// TIA Portal V17 export
// export: Created 2022-07-20T06:59:51.7556163Z, ExportSetting WithDefaults, DisplayName Totally Integrated Automation Portal, DisplayVersion V17, DisplayName TIA Portal Openness, DisplayVersion V17, DisplayName TIA Portal Version Control Interface, DisplayVersion V17, DisplayName SINAMICS Startdrive Advanced, DisplayVersion V17, DisplayName SINAMICS Startdrive G130, G150, S120, S150, SINAMICS MV, S210, DisplayVersion V17, DisplayName SINAMICS Startdrive G110M, G120, G120C, G120D, G120P, G115D, DisplayVersion V17, DisplayName STEP 7 Professional, DisplayVersion V17, DisplayName STEP 7 Safety, DisplayVersion V17, DisplayName WinCC Advanced, DisplayVersion V17
FUNCTION_BLOCK "FB10067_IperPrintingInkCircuitGen2"   // FB10067, LAD
{ S7_Optimized_Access := 'TRUE' }
VERSION : 0.1
// stored: AutoNumber false, IsIECCheckEnabled false, IsRetainMemResEnabled false, MemoryReserve 100, SetENOAutomatically false, UDAEnableTagReadback false
   VAR_INPUT
      Acknowledge : Bool;
      DegassingSystem_RisingInkSensor : Bool;
      Sensor1_Value { ExternalAccessible := 'False'; ExternalVisible := 'False'; ExternalWritable := 'False'} : Int;
      Sensor1_HighErrorThreshold { ExternalAccessible := 'False'; ExternalVisible := 'False'; ExternalWritable := 'False'} : Real;
      Sensor1_HighWarningThreshold { ExternalAccessible := 'False'; ExternalVisible := 'False'; ExternalWritable := 'False'} : Real;
      Sensor1_LowWarningThreshold { ExternalAccessible := 'False'; ExternalVisible := 'False'; ExternalWritable := 'False'} : Real;
      Sensor1_LowErrorThreshold { ExternalAccessible := 'False'; ExternalVisible := 'False'; ExternalWritable := 'False'} : Real;
      Sensor2_Value { ExternalAccessible := 'False'; ExternalVisible := 'False'; ExternalWritable := 'False'} : Int;
      Sensor2_HighErrorThreshold { ExternalAccessible := 'False'; ExternalVisible := 'False'; ExternalWritable := 'False'} : Real;
      Sensor2_HighWarningThreshold { ExternalAccessible := 'False'; ExternalVisible := 'False'; ExternalWritable := 'False'} : Real;
      Sensor2_LowWarningThreshold { ExternalAccessible := 'False'; ExternalVisible := 'False'; ExternalWritable := 'False'} : Real;
      Sensor2_LowErrorThreshold { ExternalAccessible := 'False'; ExternalVisible := 'False'; ExternalWritable := 'False'} : Real;
      BarrelWS_RawValue { ExternalAccessible := 'False'; ExternalVisible := 'False'; ExternalWritable := 'False'} : Int;
      BarrelWS_CalibrationValue_1 { ExternalAccessible := 'False'; ExternalVisible := 'False'; ExternalWritable := 'False'} : Real;
      BarrelWS_CalibrationValue_2 { ExternalAccessible := 'False'; ExternalVisible := 'False'; ExternalWritable := 'False'} : Real;
      BarrelWS_LowWarningThreshold { ExternalAccessible := 'False'; ExternalVisible := 'False'; ExternalWritable := 'False'} : Real;
      BarrelWS_HighWarningThreshold { ExternalAccessible := 'False'; ExternalVisible := 'False'; ExternalWritable := 'False'} : Real;
      BarrelWS_LowErrorThreshold { ExternalAccessible := 'False'; ExternalVisible := 'False'; ExternalWritable := 'False'} : Real;
      BarrelWS_HighErrorThreshold { ExternalAccessible := 'False'; ExternalVisible := 'False'; ExternalWritable := 'False'} : Real;
      Tank1_ReachLevel { ExternalAccessible := 'False'; ExternalVisible := 'False'; ExternalWritable := 'False'} : Real;
      Tank1_RegulationLevel { ExternalAccessible := 'False'; ExternalVisible := 'False'; ExternalWritable := 'False'} : Real;
      Tank2_ReachLevel { ExternalAccessible := 'False'; ExternalVisible := 'False'; ExternalWritable := 'False'} : Real;
      Tank2_RegulationLevel { ExternalAccessible := 'False'; ExternalVisible := 'False'; ExternalWritable := 'False'} : Real;
      SystemPressurized { ExternalAccessible := 'False'; ExternalVisible := 'False'; ExternalWritable := 'False'} : Bool;
      SystemDepressurized { ExternalAccessible := 'False'; ExternalVisible := 'False'; ExternalWritable := 'False'} : Bool;
   END_VAR
   VAR_OUTPUT
      DegassingSystem_SolenoidValve : Bool;
      DegassingSystem_RisingInkError : Bool;
      ActivePump { ExternalAccessible := 'False'; ExternalVisible := 'False'; ExternalWritable := 'False'} : Bool;
      PumpDirection { ExternalAccessible := 'False'; ExternalVisible := 'False'; ExternalWritable := 'False'} : Bool;
      ActiveGeneralSolenoid { ExternalAccessible := 'False'; ExternalVisible := 'False'; ExternalWritable := 'False'} : Bool;
      ActiveFillingSolenoid_1 { ExternalAccessible := 'False'; ExternalVisible := 'False'; ExternalWritable := 'False'} : Bool;
      ActiveFillingSolenoid_2 { ExternalAccessible := 'False'; ExternalVisible := 'False'; ExternalWritable := 'False'} : Bool;
      BarrelWS_CalibrationStatus_1 { ExternalAccessible := 'False'; ExternalVisible := 'False'; ExternalWritable := 'False'} : Bool;
      BarrelWS_CalibrationStatus_2 { ExternalAccessible := 'False'; ExternalVisible := 'False'; ExternalWritable := 'False'} : Bool;
      BarrelWS_LowWarningThresholdReached { ExternalAccessible := 'False'; ExternalVisible := 'False'; ExternalWritable := 'False'} : Bool;
      BarrelWS_HighWarningThresholdReached { ExternalAccessible := 'False'; ExternalVisible := 'False'; ExternalWritable := 'False'} : Bool;
      BarrelWS_LowErrorThresholdReached { ExternalAccessible := 'False'; ExternalVisible := 'False'; ExternalWritable := 'False'} : Bool;
      BarrelWS_HighErrorThresholdReached { ExternalAccessible := 'False'; ExternalVisible := 'False'; ExternalWritable := 'False'} : Bool;
      BarrelWS_NetWeight { ExternalAccessible := 'False'; ExternalVisible := 'False'; ExternalWritable := 'False'} : Real;
      "BarrelWS_NetWeight_%" { ExternalAccessible := 'False'; ExternalVisible := 'False'; ExternalWritable := 'False'} : Real;
      BarrelWS_CalibrationDone { ExternalAccessible := 'False'; ExternalVisible := 'False'; ExternalWritable := 'False'} : Bool;
      Tank1_VarnishQuantity_mm { ExternalAccessible := 'False'; ExternalVisible := 'False'; ExternalWritable := 'False'} : Real;
      "Tank1_VarnishQuantity_%" { ExternalAccessible := 'False'; ExternalVisible := 'False'; ExternalWritable := 'False'} : Real;
      Tank1_ReachLevelDone { ExternalAccessible := 'False'; ExternalVisible := 'False'; ExternalWritable := 'False'} : Bool;
      Tank1_AutoRegulationInProgress { ExternalAccessible := 'False'; ExternalVisible := 'False'; ExternalWritable := 'False'} : Bool;
      Tank2_VarnishQuantity_mm { ExternalAccessible := 'False'; ExternalVisible := 'False'; ExternalWritable := 'False'} : Real;
      "Tank2_VarnishQuantity_%" { ExternalAccessible := 'False'; ExternalVisible := 'False'; ExternalWritable := 'False'} : Real;
      Tank2_ReachLevelDone { ExternalAccessible := 'False'; ExternalVisible := 'False'; ExternalWritable := 'False'} : Bool;
      Tank2_AutoRegulationInProgress { ExternalAccessible := 'False'; ExternalVisible := 'False'; ExternalWritable := 'False'} : Bool;
      Sensor1_HighErrorThresholdReached { ExternalAccessible := 'False'; ExternalVisible := 'False'; ExternalWritable := 'False'} : Bool;
      Sensor1_HighWarningThresholdReached { ExternalAccessible := 'False'; ExternalVisible := 'False'; ExternalWritable := 'False'} : Bool;
      Sensor1_LowWarningThresholdReached { ExternalAccessible := 'False'; ExternalVisible := 'False'; ExternalWritable := 'False'} : Bool;
      Sensor1_LowErrorThresholdReached { ExternalAccessible := 'False'; ExternalVisible := 'False'; ExternalWritable := 'False'} : Bool;
      Sensor1_Calibrated { ExternalAccessible := 'False'; ExternalVisible := 'False'; ExternalWritable := 'False'} : Bool;
      Sensor2_HighErrorThresholdReached { ExternalAccessible := 'False'; ExternalVisible := 'False'; ExternalWritable := 'False'} : Bool;
      Sensor2_HighWarningThresholdReached { ExternalAccessible := 'False'; ExternalVisible := 'False'; ExternalWritable := 'False'} : Bool;
      Sensor2_LowWarningThresholdReached { ExternalAccessible := 'False'; ExternalVisible := 'False'; ExternalWritable := 'False'} : Bool;
      Sensor2_LowErrorThresholdReached { ExternalAccessible := 'False'; ExternalVisible := 'False'; ExternalWritable := 'False'} : Bool;
      Sensor2_Calibrated { ExternalAccessible := 'False'; ExternalVisible := 'False'; ExternalWritable := 'False'} : Bool;
      InkCircuitInError { ExternalAccessible := 'False'; ExternalVisible := 'False'; ExternalWritable := 'False'} : Bool;
      AutoRegulationPositionDeviation_1 { ExternalAccessible := 'False'; ExternalVisible := 'False'; ExternalWritable := 'False'} : Bool;
      AutoRegulationPositionDeviation_2 { ExternalAccessible := 'False'; ExternalVisible := 'False'; ExternalWritable := 'False'} : Bool;
   END_VAR
   VAR_IN_OUT
      RequestAcknowledge { ExternalAccessible := 'False'; ExternalVisible := 'False'; ExternalWritable := 'False'} : Bool;
      BarrelWS_RequestCalibration_1 { ExternalAccessible := 'False'; ExternalVisible := 'False'; ExternalWritable := 'False'} : Bool;
      BarrelWS_RequestCalibration_2 { ExternalAccessible := 'False'; ExternalVisible := 'False'; ExternalWritable := 'False'} : Bool;
      Tank1_RequestReachLevel { ExternalAccessible := 'False'; ExternalVisible := 'False'; ExternalWritable := 'False'} : Bool;
      Tank1_RequestAutoregulation { ExternalAccessible := 'False'; ExternalVisible := 'False'; ExternalWritable := 'False'} : Bool;
      Tank2_RequestReachLevel : Bool;
      Tank2_RequestAutoregulation : Bool;
      Tanks_RequestReachLevel : Bool;
      Tanks_RequestAutoregulation : Bool;
      BarrelWS_ResetCalibration { ExternalAccessible := 'False'; ExternalVisible := 'False'; ExternalWritable := 'False'} : Bool;
      Sensor1_CalibrationValueX_1 { ExternalAccessible := 'False'; ExternalVisible := 'False'; ExternalWritable := 'False'} : Real;
      Sensor1_CalibrationValueY_1 { ExternalAccessible := 'False'; ExternalVisible := 'False'; ExternalWritable := 'False'} : Real;
      Sensor1_CalibrationValueX_2 { ExternalAccessible := 'False'; ExternalVisible := 'False'; ExternalWritable := 'False'} : Real;
      Sensor1_CalibrationValueY_2 { ExternalAccessible := 'False'; ExternalVisible := 'False'; ExternalWritable := 'False'} : Real;
      Sensor2_CalibrationValueX_2 { ExternalAccessible := 'False'; ExternalVisible := 'False'; ExternalWritable := 'False'} : Real;
      Sensor2_CalibrationValueY_1 { ExternalAccessible := 'False'; ExternalVisible := 'False'; ExternalWritable := 'False'} : Real;
      Sensor2_CalibrationValueX_1 { ExternalAccessible := 'False'; ExternalVisible := 'False'; ExternalWritable := 'False'} : Real;
      Sensor2_CalibrationValueY_2 { ExternalAccessible := 'False'; ExternalVisible := 'False'; ExternalWritable := 'False'} : Real;
      BarrelWS_CalibrationDataX_1 { ExternalAccessible := 'False'; ExternalVisible := 'False'; ExternalWritable := 'False'} : Real;
      BarrelWS_CalibrationDataY_1 { ExternalAccessible := 'False'; ExternalVisible := 'False'; ExternalWritable := 'False'} : Real;
      BarrelWS_CalibrationDataX_2 { ExternalAccessible := 'False'; ExternalVisible := 'False'; ExternalWritable := 'False'} : Real;
      BarrelWS_CalibrationDataY_2 { ExternalAccessible := 'False'; ExternalVisible := 'False'; ExternalWritable := 'False'} : Real;
   END_VAR
   VAR
      DirectionSended : Bool;
      AutoRegulationReachedLevelOnce : Bool;
      AutoregulationTank1Ok : Bool;
      AutoregulationTank2Ok : Bool;
      InkTankOperationStateDiagram : Int;
      R_TRIG_RequestReachLevelTank_1 { S7_SetPoint := 'True'} : R_TRIG;
      R_TRIG_RequestReachLevelTank_2 { S7_SetPoint := 'True'} : R_TRIG;
      R_TRIG_RequestReachLevelTanks { S7_SetPoint := 'True'} : R_TRIG;
      R_TRIG_RequestAutoRegulationTank_1 { S7_SetPoint := 'True'} : R_TRIG;
      R_TRIG_RequestAutoRegulationTank_2 { S7_SetPoint := 'True'} : R_TRIG;
      R_TRIG_RequestAutoRegulationTanks { S7_SetPoint := 'True'} : R_TRIG;
      F_TRIG_RequestReachLevelTank_1 { S7_SetPoint := 'True'} : F_TRIG;
      F_TRIG_RequestReachLevelTank_2 { S7_SetPoint := 'True'} : F_TRIG;
      F_TRIG_RequestReachLevelTanks { S7_SetPoint := 'True'} : F_TRIG;
      F_TRIG_RequestAutoRegulationTank_1 { S7_SetPoint := 'True'} : F_TRIG;
      F_TRIG_RequestAutoRegulationTank_2 { S7_SetPoint := 'True'} : F_TRIG;
      F_TRIG_RequestAutoRegulationTanks { S7_SetPoint := 'True'} : F_TRIG;
      TON_AutoRegulationPositionDeviation { S7_SetPoint := 'True'} : TON_TIME;
      TON_SendActivationAfterDirection { S7_SetPoint := 'True'} : TON_TIME;
      TON_FillTankSafety { S7_SetPoint := 'True'} : TON_TIME;
      TON_OverPressure { S7_SetPoint := 'True'} : TON_TIME;
      FB10030_AnalogicalSensor_MicrosonicUltrasonicSensor_TankLevel_1 { S7_SetPoint := 'True'} : "FB10030_AnalogicalSensor";
      FB10030_AnalogicalSensor_MicrosonicUltrasonicSensor_TankLevel_2 { S7_SetPoint := 'True'} : "FB10030_AnalogicalSensor";
      FB10030_AnalogicalSensor_TLMScale_VarnishBarrel { S7_SetPoint := 'True'} : "FB10030_AnalogicalSensor";
   END_VAR
   VAR CONSTANT
      WAIT_FOR_OPERATION_REQUEST : Int := 0;
      REACH_LEVEL_TANK_1 : Int := 10;
      REACH_LEVEL_TANK_2 : Int := 20;
      REACH_LEVEL_TANKS : Int := 30;
      AUTO_REGULATION_TANK_1 : Int := 40;
      AUTO_REGULATION_TANK_2 : Int := 50;
      AUTO_REGULATION_TANKS : Int := 60;
      OPERATION_DONE : Int := 70;
   END_VAR
BEGIN

REGION Network 1 (SCL): First Scan
   IF "FirstScan" THEN
       #DirectionSended := FALSE;
       #Tank1_ReachLevelDone := FALSE;
       #Tank2_ReachLevelDone := FALSE;
       #InkTankOperationStateDiagram := #WAIT_FOR_OPERATION_REQUEST;
   END_IF;
END_REGION

REGION Network 2 (SCL): Edge Signals & Timers
   REGION EDGE SIGNALS
       #R_TRIG_RequestReachLevelTank_1(CLK := #Tank1_RequestReachLevel);
       #R_TRIG_RequestAutoRegulationTank_1(CLK := #Tank1_RequestAutoregulation);
       #R_TRIG_RequestReachLevelTank_2(CLK := #Tank1_RequestReachLevel);
       #R_TRIG_RequestAutoRegulationTank_2(CLK := #Tank2_RequestAutoregulation);
       #R_TRIG_RequestReachLevelTanks(CLK := #Tanks_RequestReachLevel);
       #R_TRIG_RequestAutoRegulationTanks(CLK := #Tanks_RequestAutoregulation);

       #F_TRIG_RequestReachLevelTank_1(CLK := #Tank1_RequestReachLevel);
       #F_TRIG_RequestAutoRegulationTank_1(CLK := #Tank1_RequestAutoregulation);
       #F_TRIG_RequestReachLevelTank_2(CLK := #Tank2_RequestReachLevel);
       #F_TRIG_RequestAutoRegulationTank_2(CLK := #Tank2_RequestAutoregulation);
       #F_TRIG_RequestReachLevelTanks(CLK := #Tanks_RequestReachLevel);
       #F_TRIG_RequestAutoRegulationTanks(CLK := #Tanks_RequestAutoregulation);
   END_REGION

   REGION TIMERS
       #TON_AutoRegulationPositionDeviation(IN := #AutoRegulationReachedLevelOnce AND NOT ("FC10021_TolerenceRelation"(X := #Tank1_VarnishQuantity_mm, Y := #Tank1_RegulationLevel, Tolerance := 10.0)),
                                            PT := T#5s);
       #TON_SendActivationAfterDirection(IN := #InkTankOperationStateDiagram = #REACH_LEVEL_TANK_1 OR
                                         #InkTankOperationStateDiagram = #REACH_LEVEL_TANK_2 OR
                                         #InkTankOperationStateDiagram = #REACH_LEVEL_TANKS OR
                                         #InkTankOperationStateDiagram = #AUTO_REGULATION_TANK_1 OR
                                         #InkTankOperationStateDiagram = #AUTO_REGULATION_TANK_2 OR
                                         #InkTankOperationStateDiagram = #AUTO_REGULATION_TANKS,
                                         PT := T#20ms); //Time direction signal sended and pump activation necessary for the electronical card
       #TON_FillTankSafety(IN := #ActivePump AND #PumpDirection,
                           PT := T#1000s);  
   END_REGION
END_REGION

REGION Network 3 (SCL): Tank Commands Management
   IF #TON_SendActivationAfterDirection.Q THEN
       #DirectionSended := TRUE;
   END_IF;
END_REGION

REGION Network 4: Ink Barrel Weigh Scale Management
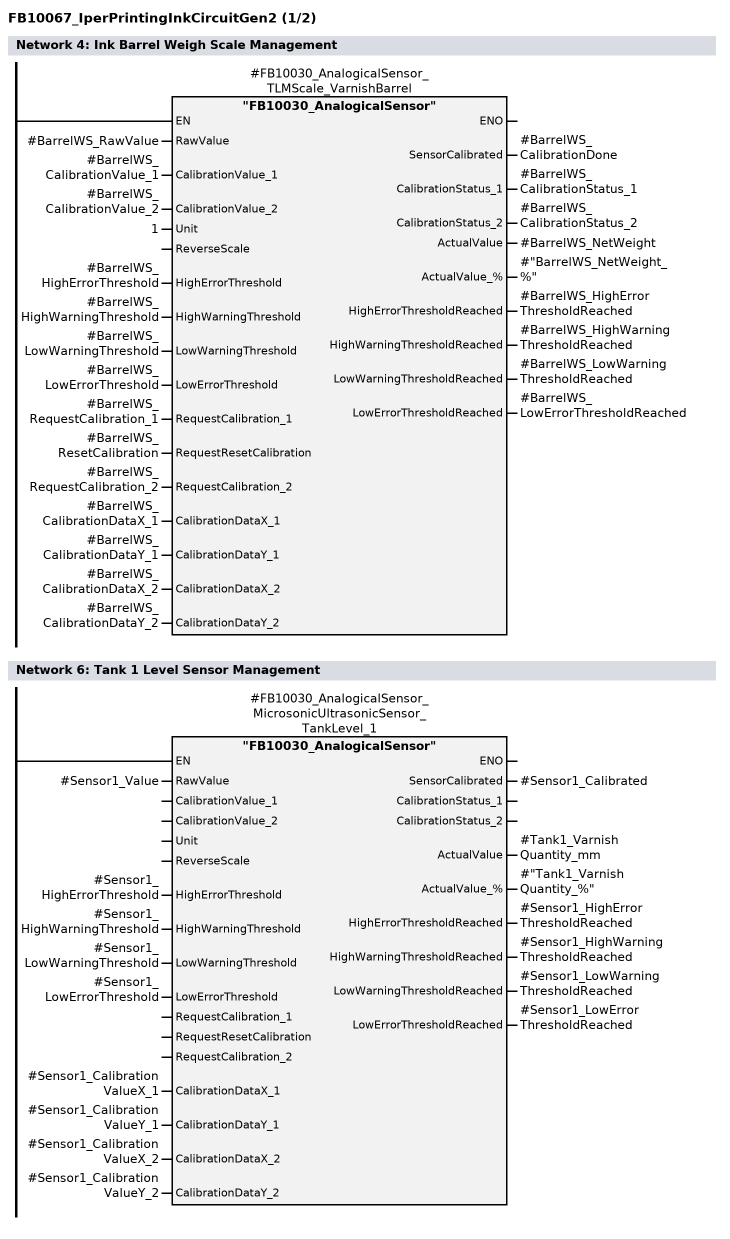
   RUNG wire#powerrail
      #FB10030_AnalogicalSensor_TLMScale_VarnishBarrel(RawValue := #BarrelWS_RawValue, CalibrationValue_1 := #BarrelWS_CalibrationValue_1, CalibrationValue_2 := #BarrelWS_CalibrationValue_2, Unit := 1, ReverseScale :=, HighErrorThreshold := #BarrelWS_HighErrorThreshold, HighWarningThreshold := #BarrelWS_HighWarningThreshold, LowWarningThreshold := #BarrelWS_LowWarningThreshold, LowErrorThreshold := #BarrelWS_LowErrorThreshold, RequestCalibration_1 := #BarrelWS_RequestCalibration_1, RequestResetCalibration := #BarrelWS_ResetCalibration, RequestCalibration_2 := #BarrelWS_RequestCalibration_2, CalibrationDataX_1 := #BarrelWS_CalibrationDataX_1, CalibrationDataY_1 := #BarrelWS_CalibrationDataY_1, CalibrationDataX_2 := #BarrelWS_CalibrationDataX_2, CalibrationDataY_2 := #BarrelWS_CalibrationDataY_2, SensorCalibrated => #BarrelWS_CalibrationDone, CalibrationStatus_1 => #BarrelWS_CalibrationStatus_1, CalibrationStatus_2 => #BarrelWS_CalibrationStatus_2, ActualValue => #BarrelWS_NetWeight, "ActualValue_%" => #"BarrelWS_NetWeight_%", HighErrorThresholdReached => #BarrelWS_HighErrorThresholdReached, HighWarningThresholdReached => #BarrelWS_HighWarningThresholdReached, LowWarningThresholdReached => #BarrelWS_LowWarningThresholdReached, LowErrorThresholdReached => #BarrelWS_LowErrorThresholdReached)
   END_RUNG
   // the same network as SCL:
   #FB10030_AnalogicalSensor_TLMScale_VarnishBarrel(RawValue := #BarrelWS_RawValue,   // "FB10030_AnalogicalSensor"
                           CalibrationValue_1 := #BarrelWS_CalibrationValue_1,
                           CalibrationValue_2 := #BarrelWS_CalibrationValue_2,
                           Unit := 1,
                           HighErrorThreshold := #BarrelWS_HighErrorThreshold,
                           HighWarningThreshold := #BarrelWS_HighWarningThreshold,
                           LowWarningThreshold := #BarrelWS_LowWarningThreshold,
                           LowErrorThreshold := #BarrelWS_LowErrorThreshold,
                           RequestCalibration_1 := #BarrelWS_RequestCalibration_1,
                           RequestResetCalibration := #BarrelWS_ResetCalibration,
                           RequestCalibration_2 := #BarrelWS_RequestCalibration_2,
                           CalibrationDataX_1 := #BarrelWS_CalibrationDataX_1,
                           CalibrationDataY_1 := #BarrelWS_CalibrationDataY_1,
                           CalibrationDataX_2 := #BarrelWS_CalibrationDataX_2,
                           CalibrationDataY_2 := #BarrelWS_CalibrationDataY_2,
                           SensorCalibrated => #BarrelWS_CalibrationDone,
                           CalibrationStatus_1 => #BarrelWS_CalibrationStatus_1,
                           CalibrationStatus_2 => #BarrelWS_CalibrationStatus_2,
                           ActualValue => #BarrelWS_NetWeight,
                           "ActualValue_%" => #"BarrelWS_NetWeight_%",
                           HighErrorThresholdReached => #BarrelWS_HighErrorThresholdReached,
                           HighWarningThresholdReached => #BarrelWS_HighWarningThresholdReached,
                           LowWarningThresholdReached => #BarrelWS_LowWarningThresholdReached,
                           LowErrorThresholdReached => #BarrelWS_LowErrorThresholdReached);
END_REGION

REGION Network 5 (SCL): Degassing System Management
   IF #DegassingSystem_RisingInkSensor THEN
       #DegassingSystem_SolenoidValve := FALSE;
       #DegassingSystem_RisingInkError := TRUE;
   ELSE
       #DegassingSystem_SolenoidValve := TRUE;
   END_IF;
END_REGION

REGION Network 6: Tank 1 Level Sensor Management
   RUNG wire#powerrail
      #FB10030_AnalogicalSensor_MicrosonicUltrasonicSensor_TankLevel_1(RawValue := #Sensor1_Value, CalibrationValue_1 :=, CalibrationValue_2 :=, Unit :=, ReverseScale :=, HighErrorThreshold := #Sensor1_HighErrorThreshold, HighWarningThreshold := #Sensor1_HighWarningThreshold, LowWarningThreshold := #Sensor1_LowWarningThreshold, LowErrorThreshold := #Sensor1_LowErrorThreshold, RequestCalibration_1 :=, RequestResetCalibration :=, RequestCalibration_2 :=, CalibrationDataX_1 := #Sensor1_CalibrationValueX_1, CalibrationDataY_1 := #Sensor1_CalibrationValueY_1, CalibrationDataX_2 := #Sensor1_CalibrationValueX_2, CalibrationDataY_2 := #Sensor1_CalibrationValueY_2, SensorCalibrated => #Sensor1_Calibrated, CalibrationStatus_1 =>, CalibrationStatus_2 =>, ActualValue => #Tank1_VarnishQuantity_mm, "ActualValue_%" => #"Tank1_VarnishQuantity_%", HighErrorThresholdReached => #Sensor1_HighErrorThresholdReached, HighWarningThresholdReached => #Sensor1_HighWarningThresholdReached, LowWarningThresholdReached => #Sensor1_LowWarningThresholdReached, LowErrorThresholdReached => #Sensor1_LowErrorThresholdReached)
   END_RUNG
   // the same network as SCL:
   #FB10030_AnalogicalSensor_MicrosonicUltrasonicSensor_TankLevel_1(RawValue := #Sensor1_Value,   // "FB10030_AnalogicalSensor"
                           HighErrorThreshold := #Sensor1_HighErrorThreshold,
                           HighWarningThreshold := #Sensor1_HighWarningThreshold,
                           LowWarningThreshold := #Sensor1_LowWarningThreshold,
                           LowErrorThreshold := #Sensor1_LowErrorThreshold,
                           CalibrationDataX_1 := #Sensor1_CalibrationValueX_1,
                           CalibrationDataY_1 := #Sensor1_CalibrationValueY_1,
                           CalibrationDataX_2 := #Sensor1_CalibrationValueX_2,
                           CalibrationDataY_2 := #Sensor1_CalibrationValueY_2,
                           SensorCalibrated => #Sensor1_Calibrated,
                           ActualValue => #Tank1_VarnishQuantity_mm,
                           "ActualValue_%" => #"Tank1_VarnishQuantity_%",
                           HighErrorThresholdReached => #Sensor1_HighErrorThresholdReached,
                           HighWarningThresholdReached => #Sensor1_HighWarningThresholdReached,
                           LowWarningThresholdReached => #Sensor1_LowWarningThresholdReached,
                           LowErrorThresholdReached => #Sensor1_LowErrorThresholdReached);
END_REGION

REGION Network 7: Tank 2 Level Sensor Management
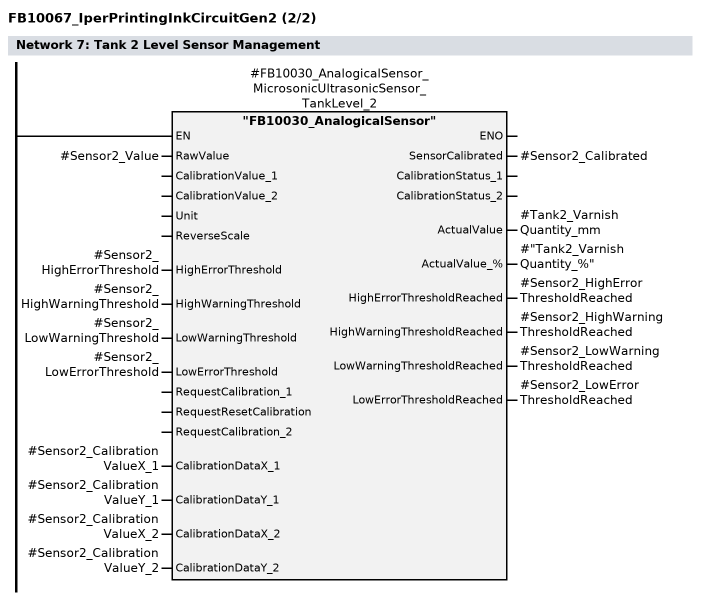
   RUNG wire#powerrail
      #FB10030_AnalogicalSensor_MicrosonicUltrasonicSensor_TankLevel_2(RawValue := #Sensor2_Value, CalibrationValue_1 :=, CalibrationValue_2 :=, Unit :=, ReverseScale :=, HighErrorThreshold := #Sensor2_HighErrorThreshold, HighWarningThreshold := #Sensor2_HighWarningThreshold, LowWarningThreshold := #Sensor2_LowWarningThreshold, LowErrorThreshold := #Sensor2_LowErrorThreshold, RequestCalibration_1 :=, RequestResetCalibration :=, RequestCalibration_2 :=, CalibrationDataX_1 := #Sensor2_CalibrationValueX_1, CalibrationDataY_1 := #Sensor2_CalibrationValueY_1, CalibrationDataX_2 := #Sensor2_CalibrationValueX_2, CalibrationDataY_2 := #Sensor2_CalibrationValueY_2, SensorCalibrated => #Sensor2_Calibrated, CalibrationStatus_1 =>, CalibrationStatus_2 =>, ActualValue => #Tank2_VarnishQuantity_mm, "ActualValue_%" => #"Tank2_VarnishQuantity_%", HighErrorThresholdReached => #Sensor2_HighErrorThresholdReached, HighWarningThresholdReached => #Sensor2_HighWarningThresholdReached, LowWarningThresholdReached => #Sensor2_LowWarningThresholdReached, LowErrorThresholdReached => #Sensor2_LowErrorThresholdReached)
   END_RUNG
   // the same network as SCL:
   #FB10030_AnalogicalSensor_MicrosonicUltrasonicSensor_TankLevel_2(RawValue := #Sensor2_Value,   // "FB10030_AnalogicalSensor"
                           HighErrorThreshold := #Sensor2_HighErrorThreshold,
                           HighWarningThreshold := #Sensor2_HighWarningThreshold,
                           LowWarningThreshold := #Sensor2_LowWarningThreshold,
                           LowErrorThreshold := #Sensor2_LowErrorThreshold,
                           CalibrationDataX_1 := #Sensor2_CalibrationValueX_1,
                           CalibrationDataY_1 := #Sensor2_CalibrationValueY_1,
                           CalibrationDataX_2 := #Sensor2_CalibrationValueX_2,
                           CalibrationDataY_2 := #Sensor2_CalibrationValueY_2,
                           SensorCalibrated => #Sensor2_Calibrated,
                           ActualValue => #Tank2_VarnishQuantity_mm,
                           "ActualValue_%" => #"Tank2_VarnishQuantity_%",
                           HighErrorThresholdReached => #Sensor2_HighErrorThresholdReached,
                           HighWarningThresholdReached => #Sensor2_HighWarningThresholdReached,
                           LowWarningThresholdReached => #Sensor2_LowWarningThresholdReached,
                           LowErrorThresholdReached => #Sensor2_LowErrorThresholdReached);
END_REGION

REGION Network 8 (SCL): Tank Ink Management
   CASE #InkTankOperationStateDiagram OF
       #WAIT_FOR_OPERATION_REQUEST:
           IF #R_TRIG_RequestReachLevelTank_1.Q OR #R_TRIG_RequestReachLevelTank_2.Q THEN
               #Tank1_ReachLevelDone := FALSE;
               #PumpDirection := TRUE;
               #InkTankOperationStateDiagram := #REACH_LEVEL_TANKS;
           ELSIF #R_TRIG_RequestAutoRegulationTank_1.Q OR #R_TRIG_RequestAutoRegulationTank_2.Q THEN
               #Tank1_ReachLevelDone := FALSE;
               #Tank2_ReachLevelDone := FALSE;
               #PumpDirection := FALSE;
               #InkTankOperationStateDiagram := #AUTO_REGULATION_TANKS;
           END_IF;
       #REACH_LEVEL_TANK_1:
           //Signals Management
           IF #DirectionSended THEN
               #ActivePump := TRUE;
               IF #Tank1_VarnishQuantity_mm >= #Tank1_ReachLevel THEN
                   #ActiveGeneralSolenoid := TRUE;
                   #ActiveFillingSolenoid_1 := TRUE;
                   #PumpDirection := FALSE;
               ELSIF #Tank1_VarnishQuantity_mm < #Tank1_ReachLevel THEN
                   #ActiveGeneralSolenoid := FALSE;
                   #ActiveFillingSolenoid_1 := TRUE;
                   #PumpDirection := TRUE;
               END_IF;
           END_IF;

           //Condition To Go To Next Step
           IF
               "FC10021_TolerenceRelation"(X := #Tank1_VarnishQuantity_mm, Y := #Tank1_ReachLevel, Tolerance := 0.1) OR
               #F_TRIG_RequestReachLevelTank_1.Q
           THEN
               #ActiveGeneralSolenoid := FALSE;
               #ActiveFillingSolenoid_1 := FALSE;
               #ActivePump := FALSE;
               #PumpDirection := FALSE;
               #Tank1_ReachLevelDone := TRUE;
               #DirectionSended := FALSE;
               RESET_TIMER(#TON_SendActivationAfterDirection);
               #InkTankOperationStateDiagram := #OPERATION_DONE;
           END_IF;
       #REACH_LEVEL_TANK_2:
           //Signals Management
           IF #DirectionSended THEN
               #ActivePump := TRUE;
               IF #Tank2_VarnishQuantity_mm >= #Tank2_ReachLevel THEN
                   #ActiveGeneralSolenoid := TRUE;
                   #ActiveFillingSolenoid_2 := TRUE;
                   #PumpDirection := FALSE;
               ELSIF #Tank2_VarnishQuantity_mm < #Tank2_ReachLevel THEN
                   #ActiveGeneralSolenoid := FALSE;
                   #ActiveFillingSolenoid_2 := TRUE;
                   #PumpDirection := TRUE;
               END_IF;
           END_IF;

           //Condition To Go To Next Step
           IF
               "FC10021_TolerenceRelation"(X := #Tank2_VarnishQuantity_mm, Y := #Tank2_ReachLevel, Tolerance := 0.1) OR
               #F_TRIG_RequestReachLevelTank_1.Q
           THEN
               #ActiveGeneralSolenoid := FALSE;
               #ActiveFillingSolenoid_2 := FALSE;
               #ActivePump := FALSE;
               #PumpDirection := FALSE;
               #Tank1_ReachLevelDone := TRUE;
               #DirectionSended := FALSE;
               RESET_TIMER(#TON_SendActivationAfterDirection);
               #InkTankOperationStateDiagram := #OPERATION_DONE;
           END_IF;
       #REACH_LEVEL_TANKS:
           //Signals Management
           IF #Tank1_RequestReachLevel AND NOT (#Tank2_RequestReachLevel) THEN
               IF #DirectionSended THEN
                   #ActivePump := TRUE;
                   IF #Tank1_VarnishQuantity_mm >= #Tank1_ReachLevel THEN
                       #ActiveGeneralSolenoid := TRUE;
                       #ActiveFillingSolenoid_1 := TRUE;
                       #ActiveFillingSolenoid_2 := FALSE;
                       #PumpDirection := FALSE;
                   ELSIF #Tank1_VarnishQuantity_mm < #Tank1_ReachLevel THEN
                       #ActiveGeneralSolenoid := FALSE;
                       #ActiveFillingSolenoid_1 := TRUE;
                       #ActiveFillingSolenoid_2 := FALSE;
                       #PumpDirection := TRUE;
                   END_IF;
               END_IF;
           ELSIF NOT (#Tank1_RequestReachLevel) AND #Tank2_RequestReachLevel THEN
               IF #DirectionSended THEN
                   #ActivePump := TRUE;
                   IF #Tank2_VarnishQuantity_mm >= #Tank2_ReachLevel THEN
                       #ActiveGeneralSolenoid := TRUE;
                       #ActiveFillingSolenoid_1 := FALSE;
                       #ActiveFillingSolenoid_2 := TRUE;
                       #PumpDirection := FALSE;
                   ELSIF #Tank2_VarnishQuantity_mm < #Tank2_ReachLevel THEN
                       #ActiveGeneralSolenoid := FALSE;
                       #ActiveFillingSolenoid_1 := FALSE;
                       #ActiveFillingSolenoid_2 := TRUE;
                       #PumpDirection := TRUE;
                   END_IF;
               END_IF;
           END_IF;

           //Condition To Go To Next Step
           IF
               (
               (
               #Tank1_RequestReachLevel AND "FC10021_TolerenceRelation"(X := #Tank1_VarnishQuantity_mm, Y := #Tank1_ReachLevel, Tolerance := 0.1) OR
               NOT(#Tank1_RequestReachLevel)
               )
               AND
               (
               #Tank2_RequestReachLevel AND "FC10021_TolerenceRelation"(X := #Tank2_VarnishQuantity_mm, Y := #Tank2_ReachLevel, Tolerance := 0.1) OR
               NOT(#Tank2_RequestReachLevel)
               )
               )
               OR
               #F_TRIG_RequestReachLevelTank_1.Q
               OR
               #F_TRIG_RequestReachLevelTank_2.Q
           THEN
               #ActiveGeneralSolenoid := FALSE;
               #ActiveFillingSolenoid_1 := FALSE;
               #ActiveFillingSolenoid_2 := FALSE;
               #ActivePump := FALSE;
               #PumpDirection := FALSE;
               #Tank1_ReachLevelDone := TRUE;
               #DirectionSended := FALSE;
               RESET_TIMER(#TON_SendActivationAfterDirection);
               #InkTankOperationStateDiagram := #OPERATION_DONE;
           END_IF;
       #AUTO_REGULATION_TANK_1:
           //Signals Management
           #Tank1_AutoRegulationInProgress := TRUE;
           IF #DirectionSended THEN
               IF #Tank1_VarnishQuantity_mm >= #Tank1_RegulationLevel THEN
                   #ActivePump := FALSE;
                   #ActiveGeneralSolenoid := FALSE;
                   #ActiveFillingSolenoid_1 := FALSE;
                   #AutoRegulationReachedLevelOnce := TRUE;
               ELSIF #Tank1_VarnishQuantity_mm < #Tank1_RegulationLevel - 1.0 THEN
                   #ActivePump := TRUE;
                   #ActiveGeneralSolenoid := FALSE;
                   #ActiveFillingSolenoid_1 := TRUE;
                   #PumpDirection := TRUE;
                   #AutoRegulationReachedLevelOnce := FALSE;
               END_IF;
           END_IF;

           //Condition To Go to Next Step
           IF #F_TRIG_RequestAutoRegulationTank_1.Q OR #TON_FillTankSafety.Q THEN
               #Tank1_AutoRegulationInProgress := FALSE;
               #ActiveGeneralSolenoid := FALSE;
               #ActiveFillingSolenoid_1 := FALSE;
               #ActivePump := FALSE;
               #PumpDirection := FALSE;
               #DirectionSended := FALSE;
               #AutoRegulationReachedLevelOnce := FALSE;
               RESET_TIMER(#TON_SendActivationAfterDirection);
               #InkTankOperationStateDiagram := #OPERATION_DONE;
           END_IF; 
       #AUTO_REGULATION_TANK_2:
           //Signals Management
           #Tank2_AutoRegulationInProgress := TRUE;
           IF #DirectionSended THEN
               IF #Tank2_VarnishQuantity_mm >= #Tank1_RegulationLevel THEN
                   #ActivePump := FALSE;
                   #ActiveGeneralSolenoid := FALSE;
                   #ActiveFillingSolenoid_2 := FALSE;
                   #AutoRegulationReachedLevelOnce := TRUE;
               ELSIF #Tank2_VarnishQuantity_mm < #Tank1_RegulationLevel - 1.0 THEN
                   #ActivePump := TRUE;
                   #ActiveGeneralSolenoid := FALSE;
                   #ActiveFillingSolenoid_2 := TRUE;
                   #PumpDirection := TRUE;
                   #AutoRegulationReachedLevelOnce := FALSE;
               END_IF;
           END_IF;

           //Condition To Go to Next Step
           IF #F_TRIG_RequestAutoRegulationTank_2.Q OR #TON_FillTankSafety.Q THEN
               #Tank1_AutoRegulationInProgress := FALSE;
               #ActiveGeneralSolenoid := FALSE;
               #ActiveFillingSolenoid_2 := FALSE;
               #ActivePump := FALSE;
               #PumpDirection := FALSE;
               #DirectionSended := FALSE;
               #AutoRegulationReachedLevelOnce := FALSE;
               RESET_TIMER(#TON_SendActivationAfterDirection);
               #InkTankOperationStateDiagram := #OPERATION_DONE;
           END_IF;
       #AUTO_REGULATION_TANKS:
           IF NOT(#AutoregulationTank1Ok) THEN
               //Signals Management
               #Tank1_AutoRegulationInProgress := TRUE;
               #Tank2_AutoRegulationInProgress := FALSE;
               IF #DirectionSended THEN
                   IF #Tank1_VarnishQuantity_mm >= #Tank1_RegulationLevel THEN
                       #ActivePump := FALSE;
                       #ActiveGeneralSolenoid := FALSE;
                       #ActiveFillingSolenoid_1 := FALSE;
                       #AutoRegulationReachedLevelOnce := TRUE;
                   ELSIF #Tank1_VarnishQuantity_mm < #Tank1_RegulationLevel - 1.0 THEN
                       #ActivePump := TRUE;
                       #ActiveGeneralSolenoid := FALSE;
                       #ActiveFillingSolenoid_1 := TRUE;
                       #PumpDirection := TRUE;
                       #AutoRegulationReachedLevelOnce := FALSE;
                   END_IF;
               END_IF;
           ELSIF NOT(#AutoregulationTank2Ok) THEN
               #Tank1_AutoRegulationInProgress := FALSE;
               #Tank2_AutoRegulationInProgress := TRUE;
               IF #DirectionSended THEN
                   IF #Tank2_VarnishQuantity_mm >= #Tank1_RegulationLevel THEN
                       #ActivePump := FALSE;
                       #ActiveGeneralSolenoid := FALSE;
                       #ActiveFillingSolenoid_2 := FALSE;
                       #AutoRegulationReachedLevelOnce := TRUE;
                   ELSIF #Tank2_VarnishQuantity_mm < #Tank1_RegulationLevel - 1.0 THEN
                       #ActivePump := TRUE;
                       #ActiveGeneralSolenoid := FALSE;
                       #ActiveFillingSolenoid_2 := TRUE;
                       #PumpDirection := TRUE;
                       #AutoRegulationReachedLevelOnce := FALSE;
                   END_IF;
               END_IF;
           END_IF;

           #AutoregulationTank1Ok := "FC10021_TolerenceRelation"(X := #Tank1_VarnishQuantity_mm, Y := #Tank1_ReachLevel, Tolerance := 0.1);
           #AutoregulationTank2Ok := "FC10021_TolerenceRelation"(X := #Tank2_VarnishQuantity_mm, Y := #Tank2_ReachLevel, Tolerance := 0.1);

           //Condition To Go to Next Step
           IF #F_TRIG_RequestAutoRegulationTanks.Q OR #TON_FillTankSafety.Q THEN
               #Tank1_AutoRegulationInProgress := FALSE;
               #Tank2_AutoRegulationInProgress := FALSE;
               #ActiveGeneralSolenoid := FALSE;
               #ActiveFillingSolenoid_1 := FALSE;
               #ActiveFillingSolenoid_2 := FALSE;
               #ActivePump := FALSE;
               #PumpDirection := FALSE;
               #DirectionSended := FALSE;
               #AutoRegulationReachedLevelOnce := FALSE;
               RESET_TIMER(#TON_SendActivationAfterDirection);
               #InkTankOperationStateDiagram := #OPERATION_DONE;
           END_IF;
       #OPERATION_DONE:
           RESET_TIMER(#TON_SendActivationAfterDirection);
           #InkTankOperationStateDiagram := #WAIT_FOR_OPERATION_REQUEST;
   END_CASE;
END_REGION

REGION Network 9 (SCL): Ink Circuit Error Management
   IF #Acknowledge THEN
       #DegassingSystem_RisingInkError := FALSE;
   END_IF;
END_REGION
END_FUNCTION_BLOCK
